(* Sets a test defined by TestName as finished. Note that the TestName-input must match
   a TestName that has been previously defined in this test suite. *)
FUNCTION TEST_FINISHED_NAMED
VAR_INPUT
    TestName : T_MaxString;
END_VAR
VAR
    Counter : UINT := 0;
    FoundTestName : BOOL := FALSE;
    FinishedAt : LWORD; // cpu cycle counter in 100ns precision
END_VAR
VAR_STAT
    FailedLookupCounter : UINT := 0;
    AlreadyPrintedFinalWarning : BOOL := FALSE;
END_VAR
VAR CONSTANT
    MaxNumberOfNonExistentTestNamesFailedLookups : UINT := 3;
END_VAR

TestName := F_LTrim(in := F_RTrim(in := TestName));
FinishedAt := F_GetCpuCounterAs64bit(GVL_TcUnit.GetCpuCounter);

(* Find the test suite and:
   1. Set the test in that test suite as finished
   2. Calculate and set the number of asserts made for that test
*)
FOR Counter := 1 TO GVL_TcUnit.NumberOfInitializedTestSuites BY 1 DO
    IF GVL_TcUnit.TestSuiteAddresses[Counter] = GVL_TcUnit.CurrentTestSuiteBeingCalled THEN
        FoundTestName := GVL_TcUnit.TestSuiteAddresses[Counter]^.SetTestFinished(TestName := TestName, FinishedAt := FinishedAt);
        IF NOT FoundTestName THEN
            IF FailedLookupCounter < MaxNumberOfNonExistentTestNamesFailedLookups THEN
                GVL_TcUnit.AdsMessageQueue.WriteLog(MsgCtrlMask := ADSLOG_MSGTYPE_ERROR,
                                                    MsgFmtStr := 'Failed to find test $'%s$'',
                                                    StrArg := TestName);
                FailedLookupCounter := FailedLookupCounter + 1;
                (* Abort TcUnit *)
                GVL_TcUnit.TcUnitRunner.AbortRunningTestSuiteTests();
            ELSIF NOT AlreadyPrintedFinalWarning THEN
                GVL_TcUnit.AdsMessageQueue.WriteLog(MsgCtrlMask := ADSLOG_MSGTYPE_ERROR,
                                                    MsgFmtStr := 'Excess failed attempts to mark test finished, failed. Further warnings will be suppressed',
                                                    StrArg := TestName);
                AlreadyPrintedFinalWarning := TRUE;
            END_IF
        ELSE
            GVL_TcUnit.TestSuiteAddresses[Counter]^.CalculateAndSetNumberOfAssertsForTest(TestName := TestName);
            GVL_TcUnit.CurrentTestIsFinished := TRUE;
        END_IF
        RETURN;
    END_IF
END_FOR

END_FUNCTION

(* stored: Version 1.1.0.1
   POU TEST_FINISHED_NAMED: Id {7a3926c3-51ee-4f1e-953f-089cfa833d72}, SpecialFunc None *)
